Staubli VAL3: fileRead.pgx

public program fileRead(string x_sTxtName)
  local bool l_bReadHead
  local num l_nRead
  local string l_sRead
  local string l_sSign[2]
  local string l_sDate[2]
  local num i
begin
  //2015.8.24
  bReadEnd=false
  bTxtHeadOk=false
  nAfterCount=0
  nApproCount=0
  nReadCount=0


  call init()
  bCycle=true
  //打开文件
  sFileName="Disk://txt/"+x_sTxtName

  //文件不存在
  if !$fileExists(sFileName)
    popUpMsg(sFileName+"文件不存在")
    logMsg(sFileName+"文件不存在")
    bCycle=false
    bCycleEnd=true
    bResumeCycle=false
    return
  endIf


  call fileClose()

  call ReadHead(nFileId,l_bReadHead,sPrdID,tPrdTool,jPrdHome,fPrdFrame,trPrdFrmOffset,nTotalTrajs)
  //判断头文件是否正确
  if l_bReadHead==false
    popUpMsg("头文件格式或内容错误")
    return
  endIf

  if nTotalTrajs!=1
    popUpMsg("路径个数不等于1")
    return
  endIf



  //关键数据核对检查
  bTxtHeadOk=true
  l_sSign[0]=""
  l_sSign[1]=""
  //
  call fileClose()
  nFileId=$fileOpen(sFileName,"r")
  //文件内容读取
  //从"BYPASS=FALSE"标示符开始采集数据
  do
    l_nRead=$fileGet(nFileId,l_sRead,1)
    //    call getStrSign(l_sRead,l_sSign)
    //    //路径结束标志
    //    if l_sSign[1]=="END"
    //      if nCurrentTraj<nTotalTrajs
    //        nCurrentTraj=nCurrentTraj+1
    //      endIf
    //    endIf
    //  until l_sSign[0]=="BYPASS" and l_sSign[1]=="FALSE"

  until find(l_sRead,"WORKPLACE=")>=0


  bBYPASS=false




  while $fileGet(nFileId,l_sRead,1)==1
    if find(l_sRead,"=END")>0
      logMsg("读取完成")
      call fileClose()
      bReadEnd=true
      return
    endIf


    if find(l_sRead,"=BEGIN")>0
      popUpMsg("程序不止一条路径")
      logMsg("读取完成")
      call fileClose()
      bReadEnd=true
      return
    endIf


    if find(l_sRead,"MOVEJ=")>=0
      if nAfterCount>99 or nApproCount>99
        popUpMsg("MOVEJ 个数不正确")
        return
      endIf
      call getStrSign(l_sRead,l_sSign)
      call getStrDate(l_sSign[1],l_sDate)
      if nReadCount==0
        call getJointDate(l_sDate[0],jJointRead[nApproCount])
        if bGetSpeed
          call getSpeedDate(l_sDate[1],mSpdOfJnt[nApproCount])
        endIf
        nApproCount=nApproCount+1

      else
        wait(nMoveCount>0)
        call getJointDate(l_sDate[0],jJointRead[nAfterCount])
        if bGetSpeed
          call getSpeedDate(l_sDate[1],mSpdOfJnt[nAfterCount])
        endIf
        nAfterCount=nAfterCount+1
      endIf

    endIf






    if find(l_sRead,"MOVEL=")>=0
      if nAfterCount!=0
        popUpMsg("文件格式不对")
        return
      endIf

      wait(nReadCount-nMoveCount<99)
      call getStrSign(l_sRead,l_sSign)
      call getStrDate(l_sSign[1],l_sDate)
      link(pPointRead[nReadCount%100],fPrdFrame)
      call getPointDate(l_sDate[0],pPointRead[nReadCount%100])
      //从TXT中获得机器人速度参数
      if bGetSpeed
        call getSpeedDate(l_sDate[1],mSpdOfPt[nReadCount%100])
      endIf
      nReadCount=nReadCount+1

    endIf


    delay(0)
  endWhile



  //  do
  //    //等待读取信息
  //    while (nReadPtr+nThousandRead*1000+900<nThousandWrite*1000+nWritePtr or nReadJnt+nHundredRead*100+50<nWriteJnt+nHundredWrite*100) and !bResumeCycle
  //      delay(0.004)
  //    endWhile
  //    l_nRead=$fileGet(nFileId,l_sRead,1)
  //    call getStrSign(l_sRead,l_sSign)
  //    //路径是否过滤
  //    if l_sSign=="BYPASS" and l_sSign[1]=="TRUE"
  //      bBYPASS=true
  //    endIf
  //    if l_sSign=="BYPASS" and l_sSign[1]=="FALSE"
  //      bBYPASS=false
  //    endIf
  //    if !bBYPASS
  //      //获取是否从TXT获得速度信息
  //      if !bGetSpeed
  //        if l_sSign=="GETSPEED" and l_sSign[1]=="TRUE"
  //          bGetSpeed=true
  //          date:libSave()
  //        endIf
  //      endIf
  //      //获取转台信息,判断模式
  //      if date:bWorTbMoving==false
  //        if l_sSign=="WORKTABLEMODE" and l_sSign[1]=="TRUE"
  //          date:bWorTbMoving=true
  //          date:libSave()
  //        endIf
  //      endIf
  //      //MOVEJ情形
  //      if l_sSign=="MOVEJ"
  //        call getStrDate(l_sSign[1],l_sDate)
  //        sMoveMode[nWritePtr]="MOVEJ"
  //        call getJointDate(l_sDate[0],jJointRead[nWriteJnt])
  //        //call getSpeedDate(l_sDate[1],mSpdOfJnt[nWriteJnt])
  //        nWriteJnt=nWriteJnt+1
  //        if nWriteJnt>99
  //          nWriteJnt=0
  //          nHundredWrite=nHundredWrite+1
  //        endIf
  //        nWritePtr=nWritePtr+1
  //        if nWritePtr>999
  //          nWritePtr=0
  //          nThousandWrite=nThousandWrite+1
  //        endIf
  //      endIf
  //      //MOVEL情形
  //      if l_sSign=="MOVEL"
  //        call getStrDate(l_sSign[1],l_sDate)
  //        sMoveMode[nWritePtr]="MOVEL"
  //        link(pPointRead[nWritePtr],fPrdFrame)
  //        call getPointDate(l_sDate[0],pPointRead[nWritePtr])
  //        //从TXT中获得机器人速度参数
  //        if bGetSpeed
  //          call getSpeedDate(l_sDate[1],mSpdOfPt[nWritePtr])
  //        endIf
  //        //          //转台转动情形
  //        //          if date:bWorTbMoving==true
  //        //            nDistToOrign=sqrt(pPointRead[nWritePtr].trsf.x*pPointRead[nWritePtr].trsf.x+pPointRead[nWritePtr].trsf.y*pPointRead[nWritePtr].trsf.y)
  //        //            //
  //        //            //修改机器人移动速度：速度关系式v=v(1-k*d/r)
  //        //            mSpdOfPt[nWritePtr].tvel=mSpdOfPt[nWritePtr].tvel*(1-0.5*nDistToOrign/nPrdRadius)
  //        //            //
  //        //          endIf
  //        nWritePtr=nWritePtr+1
  //        if nWritePtr>999
  //          nWritePtr=0
  //          nThousandWrite=nThousandWrite+1
  //        endIf
  //      endIf
  //    endIf
  //    //路径结束标志
  //    if l_sSign[1]=="END"
  //      if nCurrentTraj<nTotalTrajs
  //        if size(nPtOfTraj)<nCurrentTraj+1
  //          $dins(nPtOfTraj,size(nPtOfTraj)-1)
  //        endIf
  //        nPtOfTraj[nCurrentTraj]=nThousandWrite*1000+nWritePtr
  //        nCurrentTraj=nCurrentTraj+1
  //        l_sSign[1]=""
  //      endIf
  //    endIf
  //    delay(0)
  //  until nCurrentTraj==nTotalTrajs
  //  bWriteEnd=true
  //  $fileClose(nFileId)

  // libSave()
end
